METHOD PUBLIC MakeReferenceTo
VAR_INPUT
	ReferenceTarget : REFERENCE TO ETcVnThresholdType;
END_VAR
activeData REF= ReferenceTarget;
SetBaseDatatypeReference();
END_METHOD

PROPERTY PUBLIC Size : UDINT
GET
Size := SIZEOF(activeData);
END_GET
END_PROPERTY

METHOD TryMakeReferenceTo : BOOL
VAR_INPUT
	Target : I_Datatype;
END_VAR
VAR
	targetAsEnum : I_EnumDatatype;
	pTargetData : POINTER TO ETcVnThresholdType;
END_VAR
IF NOT Target.TryResolveAsEnumDatatype(targetAsEnum) THEN
	RETURN;
END_IF

IF targetAsEnum.Identifier <> Identifier THEN
	RETURN;
END_IF

pTargetData := Target.Address;
activeData REF= pTargetData^;
SetBaseDatatypeReference();
TryMakeReferenceTo := TRUE;
END_METHOD

PROPERTY PUBLIC Value : ETcVnThresholdType
GET
Value := activeData;
END_GET
SET
activeData := Value;
END_SET
END_PROPERTY

END_FUNCTION_BLOCK

// Datatypes/Enums/_ETcVnVectorCompareMethod
{attribute 'linkalways'} 
{attribute 'no_explicit_call' := 'This FB is a CLASS and must be accessed using methods or properties'}
{attribute 'enable_dynamic_creation'}
FUNCTION_BLOCK _ETcVnVectorCompareMethod EXTENDS EnumDatatypeBase
VAR
	localData : ETcVnVectorCompareMethod;
	activeData : REFERENCE TO ETcVnVectorCompareMethod;
	enumBaseDatatype : _DINT(localData);
END_VAR

METHOD FB_init : BOOL
VAR_INPUT
	bInitRetains : BOOL; // if TRUE, the retain variables are initialized (warm start / cold start)
	bInCopyCode : BOOL;  // if TRUE, the instance afterwards gets moved into the copy code (online change)
	InitialValue : ETcVnVectorCompareMethod;
END_VAR
localData := InitialValue;
AddBaseDatatype(enumBaseDatatype);
ClearReference();

AddLocalEnumeration('TCVN_VCM_EUCLIDEAN', ETcVnVectorCompareMethod.TCVN_VCM_EUCLIDEAN);
AddLocalEnumeration('TCVN_VCM_ELEMENTWISE', ETcVnVectorCompareMethod.TCVN_VCM_ELEMENTWISE);
END_METHOD

METHOD PRIVATE AddLocalEnumeration
VAR_INPUT
	Enumeration : T_MAXSTRING;
	Value : ETcVnVectorCompareMethod;
END_VAR
AddEnumeration(Enumeration, Value);
END_METHOD

METHOD IsEnumeratorValueEqual : BOOL
VAR_INPUT
	Enumerator : I_KeyValueForwardEnumerator;
END_VAR
VAR
	storedValue : ETcVnVectorCompareMethod;
END_VAR
IF NOT Enumerator.TryGet(storedValue) THEN
	RETURN;
END_IF

IsEnumeratorValueEqual := storedValue = activeData;
END_METHOD

METHOD PROTECTED SetBaseDatatypeReference
VAR_INPUT
END_VAR
enumBaseDatatype.MakeReferenceTo(activeData);
END_METHOD

PROPERTY PUBLIC Address : PVOID
GET
Address := ADR(activeData);
END_GET
END_PROPERTY

METHOD PUBLIC ClearReference
VAR_INPUT
END_VAR
activeData REF= localData;
SetBaseDatatypeReference();
END_METHOD

METHOD PUBLIC Clone : I_Datatype
VAR
    pClone : POINTER TO _ETcVnVectorCompareMethod;
END_VAR
pClone := __NEW(_ETcVnVectorCompareMethod(InitialValue := Value));
Clone := pClone^;
END_METHOD

PROPERTY PUBLIC Identifier : T_MAXSTRING
GET
Identifier := 'ETcVnVectorCompareMethod';
END_GET
END_PROPERTY

METHOD PUBLIC MakeReferenceTo
VAR_INPUT
	ReferenceTarget : REFERENCE TO ETcVnVectorCompareMethod;
END_VAR
activeData REF= ReferenceTarget;
SetBaseDatatypeReference();
END_METHOD

PROPERTY PUBLIC Size : UDINT
GET
Size := SIZEOF(activeData);
END_GET
END_PROPERTY

METHOD TryMakeReferenceTo : BOOL
VAR_INPUT
	Target : I_Datatype;
END_VAR
VAR
	targetAsEnum : I_EnumDatatype;
	pTargetData : POINTER TO ETcVnVectorCompareMethod;
END_VAR
IF NOT Target.TryResolveAsEnumDatatype(targetAsEnum) THEN
	RETURN;
END_IF

IF targetAsEnum.Identifier <> Identifier THEN
	RETURN;
END_IF

pTargetData := Target.Address;
activeData REF= pTargetData^;
SetBaseDatatypeReference();
TryMakeReferenceTo := TRUE;
END_METHOD

PROPERTY PUBLIC Value : ETcVnVectorCompareMethod
GET
Value := activeData;
END_GET
SET
activeData := Value;
END_SET
END_PROPERTY

END_FUNCTION_BLOCK

// Datatypes/Enums/_ETcVnWorldCoordinateSystem
{attribute 'linkalways'} 
{attribute 'no_explicit_call' := 'This FB is a CLASS and must be accessed using methods or properties'}
{attribute 'enable_dynamic_creation'}
FUNCTION_BLOCK _ETcVnWorldCoordinateSystem EXTENDS EnumDatatypeBase
VAR
	localData : ETcVnWorldCoordinateSystem;
	activeData : REFERENCE TO ETcVnWorldCoordinateSystem;
	enumBaseDatatype : _DINT(localData);
END_VAR

METHOD FB_init : BOOL
VAR_INPUT
	bInitRetains : BOOL; // if TRUE, the retain variables are initialized (warm start / cold start)
	bInCopyCode : BOOL;  // if TRUE, the instance afterwards gets moved into the copy code (online change)
	InitialValue : ETcVnWorldCoordinateSystem;
END_VAR
localData := InitialValue;
AddBaseDatatype(enumBaseDatatype);
ClearReference();

AddLocalEnumeration('TCVN_WCS_X_RIGHT_Y_DOWN' , ETcVnWorldCoordinateSystem.TCVN_WCS_X_RIGHT_Y_DOWN);
AddLocalEnumeration('TCVN_WCS_X_DOWN_Y_RIGHT', ETcVnWorldCoordinateSystem.TCVN_WCS_X_DOWN_Y_RIGHT);
AddLocalEnumeration('TCVN_WCS_X_LEFT_Y_DOWN', ETcVnWorldCoordinateSystem.TCVN_WCS_X_LEFT_Y_DOWN);
AddLocalEnumeration('TCVN_WCS_X_UP_Y_RIGHT', ETcVnWorldCoordinateSystem.TCVN_WCS_X_UP_Y_RIGHT);
AddLocalEnumeration('TCVN_WCS_X_RIGHT_Y_UP', ETcVnWorldCoordinateSystem.TCVN_WCS_X_RIGHT_Y_UP);
AddLocalEnumeration('TCVN_WCS_X_DOWN_Y_LEFT', ETcVnWorldCoordinateSystem.TCVN_WCS_X_DOWN_Y_LEFT);
AddLocalEnumeration('TCVN_WCS_X_LEFT_Y_UP', ETcVnWorldCoordinateSystem.TCVN_WCS_X_LEFT_Y_UP);
AddLocalEnumeration('TCVN_WCS_X_UP_Y_LEFT', ETcVnWorldCoordinateSystem.TCVN_WCS_X_UP_Y_LEFT);
END_METHOD

METHOD PRIVATE AddLocalEnumeration
VAR_INPUT
	Enumeration : T_MAXSTRING;
	Value : ETcVnWorldCoordinateSystem;
END_VAR
AddEnumeration(Enumeration, Value);
END_METHOD

METHOD IsEnumeratorValueEqual : BOOL
VAR_INPUT
	Enumerator : I_KeyValueForwardEnumerator;
END_VAR
VAR
	storedValue : ETcVnWorldCoordinateSystem;
END_VAR
IF NOT Enumerator.TryGet(storedValue) THEN
	RETURN;
END_IF

IsEnumeratorValueEqual := storedValue = activeData;
END_METHOD

METHOD PROTECTED SetBaseDatatypeReference
VAR_INPUT
END_VAR
enumBaseDatatype.MakeReferenceTo(activeData);
END_METHOD

PROPERTY PUBLIC Address : PVOID
GET
Address := ADR(activeData);
END_GET
END_PROPERTY

METHOD PUBLIC ClearReference
VAR_INPUT
END_VAR
activeData REF= localData;
SetBaseDatatypeReference();
END_METHOD

METHOD PUBLIC Clone : I_Datatype
VAR
    pClone : POINTER TO _ETcVnWorldCoordinateSystem;
END_VAR
pClone := __NEW(_ETcVnWorldCoordinateSystem(InitialValue := Value));
Clone := pClone^;
END_METHOD

PROPERTY PUBLIC Identifier : T_MAXSTRING
GET
Identifier := 'ETcVnWorldCoordinateSystem';
END_GET
END_PROPERTY

METHOD PUBLIC MakeReferenceTo
VAR_INPUT
	ReferenceTarget : REFERENCE TO ETcVnWorldCoordinateSystem;
END_VAR
activeData REF= ReferenceTarget;
SetBaseDatatypeReference();
END_METHOD

PROPERTY PUBLIC Size : UDINT
GET
Size := SIZEOF(activeData);
END_GET
END_PROPERTY

METHOD TryMakeReferenceTo : BOOL
VAR_INPUT
	Target : I_Datatype;
END_VAR
VAR
	targetAsEnum : I_EnumDatatype;
	pTargetData : POINTER TO ETcVnWorldCoordinateSystem;
END_VAR
IF NOT Target.TryResolveAsEnumDatatype(targetAsEnum) THEN
	RETURN;
END_IF

IF targetAsEnum.Identifier <> Identifier THEN
	RETURN;
END_IF

pTargetData := Target.Address;
activeData REF= pTargetData^;
SetBaseDatatypeReference();
TryMakeReferenceTo := TRUE;
END_METHOD

PROPERTY PUBLIC Value : ETcVnWorldCoordinateSystem
GET
Value := activeData;
END_GET
SET
activeData := Value;
END_SET
END_PROPERTY

END_FUNCTION_BLOCK

// Datatypes/Enums/_ETcWatchdogAccumulationType
{attribute 'linkalways'} 
{attribute 'no_explicit_call' := 'This FB is a CLASS and must be accessed using methods or properties'}
{attribute 'enable_dynamic_creation'}
FUNCTION_BLOCK _ETcWatchdogAccumulationType EXTENDS EnumDatatypeBase
VAR
	localData : ETcWatchdogAccumulationType;
	activeData : REFERENCE TO ETcWatchdogAccumulationType;
	enumBaseDatatype : _UINT(localData);
END_VAR

METHOD FB_init : BOOL
VAR_INPUT
	bInitRetains : BOOL; // if TRUE, the retain variables are initialized (warm start / cold start)
	bInCopyCode : BOOL;  // if TRUE, the instance afterwards gets moved into the copy code (online change)
	InitialValue : ETcWatchdogAccumulationType;
END_VAR
localData := InitialValue;
AddBaseDatatype(enumBaseDatatype);
ClearReference();

AddLocalEnumeration('WD_ACC_TYPE_MEAN', ETcWatchdogAccumulationType.WD_ACC_TYPE_MEAN);
AddLocalEnumeration('WD_ACC_TYPE_PRODUCT', ETcWatchdogAccumulationType.WD_ACC_TYPE_PRODUCT);
END_METHOD

METHOD PRIVATE AddLocalEnumeration
VAR_INPUT
	Enumeration : T_MAXSTRING;
	Value : ETcWatchdogAccumulationType;
END_VAR
AddEnumeration(Enumeration, Value);
END_METHOD

METHOD IsEnumeratorValueEqual : BOOL
VAR_INPUT
	Enumerator : I_KeyValueForwardEnumerator;
END_VAR
VAR
	storedValue : ETcWatchdogAccumulationType;
END_VAR
IF NOT Enumerator.TryGet(storedValue) THEN
	RETURN;
END_IF

IsEnumeratorValueEqual := storedValue = activeData;
END_METHOD

METHOD PROTECTED SetBaseDatatypeReference
VAR_INPUT
END_VAR
enumBaseDatatype.MakeReferenceTo(activeData);
END_METHOD

PROPERTY PUBLIC Address : PVOID
GET
Address := ADR(activeData);
END_GET
END_PROPERTY

METHOD PUBLIC ClearReference
VAR_INPUT
END_VAR
activeData REF= localData;
SetBaseDatatypeReference();
END_METHOD

METHOD PUBLIC Clone : I_Datatype
VAR
    pClone : POINTER TO _ETcWatchdogAccumulationType;
END_VAR
pClone := __NEW(_ETcWatchdogAccumulationType(InitialValue := Value));
Clone := pClone^;
END_METHOD

PROPERTY PUBLIC Identifier : T_MAXSTRING
GET
Identifier := 'ETcWatchdogAccumulationType';
END_GET
END_PROPERTY

METHOD PUBLIC MakeReferenceTo
VAR_INPUT
	ReferenceTarget : REFERENCE TO ETcWatchdogAccumulationType;
END_VAR
activeData REF= ReferenceTarget;
SetBaseDatatypeReference();
END_METHOD

PROPERTY PUBLIC Size : UDINT
GET
Size := SIZEOF(activeData);
END_GET
END_PROPERTY

METHOD TryMakeReferenceTo : BOOL
VAR_INPUT
	Target : I_Datatype;
END_VAR
VAR
	targetAsEnum : I_EnumDatatype;
	pTargetData : POINTER TO ETcWatchdogAccumulationType;
END_VAR
IF NOT Target.TryResolveAsEnumDatatype(targetAsEnum) THEN
	RETURN;
END_IF

IF targetAsEnum.Identifier <> Identifier THEN
	RETURN;
END_IF

pTargetData := Target.Address;
activeData REF= pTargetData^;
SetBaseDatatypeReference();
TryMakeReferenceTo := TRUE;
END_METHOD

PROPERTY PUBLIC Value : ETcWatchdogAccumulationType
GET
Value := activeData;
END_GET
SET
activeData := Value;
END_SET
END_PROPERTY

END_FUNCTION_BLOCK

// Datatypes/Enums/_GEV_CAMERA_STATE
{attribute 'linkalways'} 
{attribute 'no_explicit_call' := 'This FB is a CLASS and must be accessed using methods or properties'}
{attribute 'enable_dynamic_creation'}
FUNCTION_BLOCK _GEV_CAMERA_STATE EXTENDS EnumDatatypeBase
VAR
	localData : GEV_CAMERA_STATE;
	activeData : REFERENCE TO GEV_CAMERA_STATE;
	enumBaseDatatype : _BYTE(localData);
END_VAR

METHOD FB_init : BOOL
VAR_INPUT
	bInitRetains : BOOL; // if TRUE, the retain variables are initialized (warm start / cold start)
	bInCopyCode : BOOL;  // if TRUE, the instance afterwards gets moved into the copy code (online change)
	InitialValue : GEV_CAMERA_STATE;
END_VAR
localData := InitialValue;
AddBaseDatatype(enumBaseDatatype);
ClearReference();

AddLocalEnumeration('GEV_CAMERA_IDLE', GEV_CAMERA_STATE.GEV_CAMERA_IDLE);
AddLocalEnumeration('GEV_CONTROL_CHANNEL_OPEN_MASK', GEV_CAMERA_STATE.GEV_CONTROL_CHANNEL_OPEN_MASK);
AddLocalEnumeration('GEV_STREAM_CHANNELS_OPEN_MASK', GEV_CAMERA_STATE.GEV_STREAM_CHANNELS_OPEN_MASK);
AddLocalEnumeration('GEV_CONTROL_CHANNEL_OPEN', GEV_CAMERA_STATE.GEV_CONTROL_CHANNEL_OPEN);
AddLocalEnumeration('GEV_STREAM_CHANNELS_OPEN', GEV_CAMERA_STATE.GEV_STREAM_CHANNELS_OPEN);
END_METHOD

METHOD PRIVATE AddLocalEnumeration
VAR_INPUT
	Enumeration : T_MAXSTRING;
	Value : GEV_CAMERA_STATE;
END_VAR
AddEnumeration(Enumeration, Value);
END_METHOD

METHOD IsEnumeratorValueEqual : BOOL
VAR_INPUT
	Enumerator : I_KeyValueForwardEnumerator;
END_VAR
VAR
	storedValue : GEV_CAMERA_STATE;
END_VAR
IF NOT Enumerator.TryGet(storedValue) THEN
	RETURN;
END_IF

IsEnumeratorValueEqual := storedValue = activeData;
END_METHOD

METHOD PROTECTED SetBaseDatatypeReference
VAR_INPUT
END_VAR
enumBaseDatatype.MakeReferenceTo(activeData);
END_METHOD

PROPERTY PUBLIC Address : PVOID
GET
Address := ADR(activeData);
END_GET
END_PROPERTY

METHOD PUBLIC ClearReference
VAR_INPUT
END_VAR
activeData REF= localData;
SetBaseDatatypeReference();
END_METHOD

METHOD PUBLIC Clone : I_Datatype
VAR
    pClone : POINTER TO _GEV_CAMERA_STATE;
END_VAR
pClone := __NEW(_GEV_CAMERA_STATE(InitialValue := Value));
Clone := pClone^;
END_METHOD

PROPERTY PUBLIC Identifier : T_MAXSTRING
GET
Identifier := 'GEV_CAMERA_STATE';
END_GET
END_PROPERTY

METHOD PUBLIC MakeReferenceTo
VAR_INPUT
	ReferenceTarget : REFERENCE TO GEV_CAMERA_STATE;
END_VAR
activeData REF= ReferenceTarget;
SetBaseDatatypeReference();
END_METHOD

PROPERTY PUBLIC Size : UDINT
GET
Size := SIZEOF(activeData);
END_GET
END_PROPERTY

METHOD TryMakeReferenceTo : BOOL
VAR_INPUT
	Target : I_Datatype;
END_VAR
VAR
	targetAsEnum : I_EnumDatatype;
	pTargetData : POINTER TO GEV_CAMERA_STATE;
END_VAR
IF NOT Target.TryResolveAsEnumDatatype(targetAsEnum) THEN
	RETURN;
END_IF

IF targetAsEnum.Identifier <> Identifier THEN
	RETURN;
END_IF

pTargetData := Target.Address;
activeData REF= pTargetData^;
SetBaseDatatypeReference();
TryMakeReferenceTo := TRUE;
END_METHOD

PROPERTY PUBLIC Value : GEV_CAMERA_STATE
GET
Value := activeData;
END_GET
SET
activeData := Value;
END_SET
END_PROPERTY

END_FUNCTION_BLOCK

// Datatypes/Interface/_ITcVnImage
{attribute 'linkalways'} 
{attribute 'no_explicit_call' := 'This FB is a CLASS and must be accessed using methods or properties'}
{attribute 'enable_dynamic_creation'}
FUNCTION_BLOCK _ITcVnImage EXTENDS InterfaceDatatypeBase
VAR
	localData : ITcVnImage;
	activeData : REFERENCE TO ITcVnImage REF= localData;
END_VAR

METHOD PRIVATE TryGetElementTypeFromInfo : BOOL;
VAR_INPUT
	ImageInfo : TcVnImageInfo;
	Destination : REFERENCE TO ETcVnElementType;
END_VAR
CASE ImageInfo.stPixelFormat.nElementSize OF
	
	8 : // 8bit
	
		IF ImageInfo.stPixelFormat.bSigned THEN
			Destination := ETcVnElementType.TCVN_ET_SINT;
		ELSE	
			Destination := ETcVnElementType.TCVN_ET_USINT;
		END_IF
		TryGetElementTypeFromInfo := TRUE;
	
	16 : // 16bit
	
		IF ImageInfo.stPixelFormat.bSigned THEN
			Destination := ETcVnElementType.TCVN_ET_INT;
		ELSE	
			Destination := ETcVnElementType.TCVN_ET_UINT;
		END_IF
		TryGetElementTypeFromInfo := TRUE;
	
	32 : // 32bit
	
		IF ImageInfo.stPixelFormat.bSigned AND NOT ImageInfo.stPixelFormat.bFloat THEN
			Destination := ETcVnElementType.TCVN_ET_DINT;
			TryGetElementTypeFromInfo := TRUE;
		END_IF
		
		IF ImageInfo.stPixelFormat.bFloat THEN
			Destination := ETcVnElementType.TCVN_ET_REAL;
			TryGetElementTypeFromInfo := TRUE;
		END_IF
		
	64 : // 64bit
	
		IF ImageInfo.stPixelFormat.bFloat THEN
			Destination := ETcVnElementType.TCVN_ET_LREAL;
			TryGetElementTypeFromInfo := TRUE;
		END_IF
		
ELSE
	
	RETURN;

END_CASE
END_METHOD

PROPERTY PUBLIC Address : PVOID
GET
Address := ADR(activeData);
END_GET
END_PROPERTY

METHOD PUBLIC ClearReference
VAR_INPUT
END_VAR
activeData REF= localData;
END_METHOD

METHOD PUBLIC Clone : I_Datatype
VAR
    pClone : POINTER TO _ITcVnImage;
END_VAR
pClone := __NEW(_ITcVnImage);
Clone := pClone^;
END_METHOD

PROPERTY PUBLIC Identifier : T_MAXSTRING
GET
Identifier := 'ITcVnImage';
END_GET
END_PROPERTY

METHOD PUBLIC MakeReferenceTo
VAR_INPUT
	ReferenceTarget : REFERENCE TO ITcVnImage;
END_VAR
activeData REF= ReferenceTarget;
END_METHOD

METHOD PUBLIC SerializeWith
VAR_INPUT
	Serializer : I_Serializer;
END_VAR
VAR
	result: HRESULT;
	exportImageSize: ULINT;
	buffer : POINTER TO BYTE;
	imageInfo : _TcVnImageInfo;
END_VAR
IF NOT (activeData <> 0) THEN
	// no image available, so drop out.. need to add serialization?
	Serializer.AddNull();
	RETURN;
END_IF

result := F_VN_ExportImageSize(ipImage:=activeData, nBufferSize:=exportImageSize, hrPrev:=result);

IF FAILED(result) THEN
	// export to bmp size failed, so drop out.. need to add serialization?
	Serializer.AddNull();
	RETURN;
END_IF

IF exportImageSize > DatatypeLimits.UDINT_MAX_VALUE THEN
	// export is too big for __NEW, so drop out..
	Serializer.AddNull();
	RETURN;
END_IF

IF exportImageSize <= 0 THEN
	// export is zero size, so drop out.. 
	Serializer.AddNull();
	RETURN;
END_IF
	
buffer := __NEW(BYTE,ULINT_TO_UDINT(exportImageSize));
result := F_VN_ExportImage(ipImage:=activeData, pBuffer:=buffer, nBufferSize:=exportImageSize, hrPrev:=result);

IF FAILED(result) THEN
	// export to bmp failed, so drop out.. 
	Serializer.AddNull();
	__DELETE(buffer);
	RETURN;
END_IF

activeData.GetImageInfo(imageInfo.value);

Serializer.StartObject();
Serializer.AddKeyObject('imageInfo',imageInfo);
Serializer.AddKey('imageData');
Serializer.AddBase64(buffer,ULINT_TO_DINT(exportImageSize));
Serializer.EndObject();

__DELETE(buffer);
END_METHOD

PROPERTY PUBLIC Size : UDINT
GET
Size := SIZEOF(activeData);
END_GET
END_PROPERTY

METHOD TryDeserializeFrom : BOOL
VAR_INPUT
	Deserializer : I_Deserializer;
	Feedback : I_DeserializerFeedback;
END_VAR
VAR
	imageInfo : _TcVnImageInfo;
	imageSizeInBytes : UDINT;
	buffer : POINTER TO BYTE;
	hr : HRESULT;
	elementType : ETcVnElementType;
END_VAR
IF NOT Deserializer.TryDeserializeKeyToObject('imageInfo', imageInfo, Feedback) THEN
	RETURN;
END_IF

imageSizeInBytes := ULINT_TO_UDINT(imageInfo.nImageSize.Value);

IF imageSizeInBytes = 0 THEN
	TryDeserializeFrom := TRUE;
	RETURN;
END_IF

buffer := __NEW(BYTE, imageSizeInBytes);

IF NOT Deserializer.TryGetKeyBase64('imageData', buffer, imageSizeInBytes, Feedback) THEN
	__DELETE(buffer);
	RETURN;
END_IF

TryGetElementTypeFromInfo(imageInfo.Value, elementType);

hr := F_VN_CreateImageFromArray(
	pData := buffer,
	ipImage := activeData,
	nWidth := imageInfo.nWidth.Value,
	nHeight :=  imageInfo.nHeight.Value,
	ePixelType := elementType,
	nChannelNum := imageInfo.stPixelFormat.nChannels.Value, 
	hrPrev := hr);

__DELETE(buffer);

TryDeserializeFrom := TRUE;
END_METHOD

METHOD TryMakeReferenceTo : BOOL
VAR_INPUT
	Target : I_Datatype;
END_VAR
VAR
	targetAsInterface : I_InterfaceDatatype;
	pTargetData : POINTER TO ITcVnImage;
END_VAR
IF NOT Target.TryResolveAsInterfaceDatatype(targetAsInterface) THEN
	RETURN;
END_IF

IF targetAsInterface.Identifier <> Identifier THEN
	RETURN;
END_IF

pTargetData := Target.Address;
activeData REF= pTargetData^;
TryMakeReferenceTo := TRUE;
END_METHOD

PROPERTY PUBLIC Value : REFERENCE TO ITcVnImage
GET
Value REF= activeData;
END_GET
END_PROPERTY

END_FUNCTION_BLOCK

// Datatypes/Structs/_TcVnImageInfo
{attribute 'linkalways'} 
{attribute 'no_explicit_call' := 'This FB is a CLASS and must be accessed using methods or properties'}
{attribute 'enable_dynamic_creation'}
FUNCTION_BLOCK _TcVnImageInfo EXTENDS StructuredDatatypeBase
VAR
	localData : TcVnImageInfo;
	activeData : REFERENCE TO TcVnImageInfo REF= localData;
	_nImageSize : _ULINT(localData.nImageSize);
	_nWidth : _UDINT(localData.nWidth);
	_nHeight : _UDINT(localData.nHeight);
	_nXPadding : _UINT(localData.nXPadding);
	_nYPadding : _UINT(localData.nYPadding);
	_stPixelFormat : _TcVnPixelFormat();
END_VAR

METHOD FB_init : BOOL
VAR_INPUT
	bInitRetains : BOOL; // if TRUE, the retain variables are initialized (warm start / cold start)
	bInCopyCode : BOOL;  // if TRUE, the instance afterwards gets moved into the copy code (online change)
END_VAR
SetMemberReference();
AddMember('nImageSize',_nImageSize);
AddMember('nWidth',_nWidth);
AddMember('nHeight',_nHeight);
AddMember('nXPadding',_nXPadding);
AddMember('nYPadding',_nYPadding);
AddMember('stPixelFormat',_stPixelFormat);
END_METHOD

METHOD PROTECTED SetMemberReference
VAR_INPUT
END_VAR
_nImageSize.MakeReferenceTo(activeData.nImageSize);
_nWidth.MakeReferenceTo(activeData.nWidth);
_nHeight.MakeReferenceTo(activeData.nHeight);
_nXPadding.MakeReferenceTo(activeData.nXPadding);
_nYPadding.MakeReferenceTo(activeData.nYPadding);
_stPixelFormat.MakeReferenceTo(activeData.stPixelFormat);
END_METHOD

PROPERTY PUBLIC Address : PVOID
GET
Address := ADR(activeData);
END_GET
END_PROPERTY

METHOD PUBLIC ClearReference
VAR_INPUT
END_VAR
activeData REF= localData;
SetMemberReference();
END_METHOD

METHOD PUBLIC Clone : I_Datatype
VAR
    pClone : POINTER TO _TcVnImageInfo;
END_VAR
pClone := __NEW(_TcVnImageInfo());
pClone^.Value := Value;
Clone := pClone^;
END_METHOD

PROPERTY PUBLIC Identifier : T_MAXSTRING
GET
Identifier := 'TcVnImageInfo';
END_GET
END_PROPERTY

METHOD PUBLIC MakeReferenceTo
VAR_INPUT
	ReferenceTarget : REFERENCE TO TcVnImageInfo;
END_VAR
activeData REF= ReferenceTarget;
SetMemberReference();
END_METHOD

PROPERTY PUBLIC nHeight : Reference to _UDINT
GET
nHeight REF= _nHeight;
END_GET
END_PROPERTY

PROPERTY PUBLIC nImageSize : Reference to _ULINT
GET
nImageSize REF= _nImageSize;
END_GET
END_PROPERTY

PROPERTY PUBLIC nWidth : Reference to _UDINT
GET
nWidth REF= _nWidth;
END_GET
END_PROPERTY

PROPERTY PUBLIC nXPadding : Reference to _UINT
GET
nXPadding REF= _nXPadding;
END_GET
END_PROPERTY

PROPERTY PUBLIC nYPadding : Reference to _UINT
GET
nYPadding REF= _nYPadding;
END_GET
END_PROPERTY

PROPERTY PUBLIC Size : UDINT
GET
Size := SIZEOF(activeData);
END_GET
END_PROPERTY

PROPERTY PUBLIC stPixelFormat : Reference to _TcVnPixelFormat
GET
stPixelFormat REF= _stPixelFormat;
END_GET
END_PROPERTY

METHOD TryMakeReferenceTo : BOOL
VAR_INPUT
	Target : I_Datatype;
END_VAR
VAR
	targetAsStruct : I_StructuredDatatype;
	pTargetData : POINTER TO TcVnImageInfo;
END_VAR
IF NOT Target.TryResolveAsStructuredDatatype(targetAsStruct) THEN
	RETURN;
END_IF

IF NOT (targetAsStruct.Identifier = Identifier) THEN
	RETURN;
END_IF

pTargetData := Target.Address;
activeData REF= pTargetData^;
SetMemberReference();
TryMakeReferenceTo := TRUE;
END_METHOD

PROPERTY PUBLIC Value : reference to TcVnImageInfo
GET
Value ref= activeData;
END_GET
END_PROPERTY

END_FUNCTION_BLOCK

// Datatypes/Structs/_TcVnPixelFormat
{attribute 'linkalways'} 
{attribute 'no_explicit_call' := 'This FB is a CLASS and must be accessed using methods or properties'}
{attribute 'enable_dynamic_creation'}
FUNCTION_BLOCK _TcVnPixelFormat EXTENDS StructuredDatatypeBase
VAR
	localData : TcVnPixelFormat;
	activeData : REFERENCE TO TcVnPixelFormat REF= localData;

	_bSupported : _BIT();
	_bSigned : _BIT();
	_bPlanar : _BIT();
	_bFloat : _BIT();
	_nChannels : _BYTE(localData.nChannels);
	_ePixelEncoding : _ETcVnPixelEncoding(localData.ePixelEncoding);
	_ePixelPackMode : _ETcVnPixelPackMode(localData.ePixelPackMode);
	_nElementSize : _UINT(localData.nElementSize);
	_nTotalSize : _UINT(localData.nTotalSize);
END_VAR

METHOD FB_init : BOOL
VAR_INPUT
	bInitRetains : BOOL; // if TRUE, the retain variables are initialized (warm start / cold start)
	bInCopyCode : BOOL;  // if TRUE, the instance afterwards gets moved into the copy code (online change)
END_VAR
SetMemberReference();
AddMember('bSupported',_bSupported);
AddMember('bSigned',_bSigned);
AddMember('bPlanar',_bPlanar);
AddMember('bFloat',_bFloat);
AddMember('nChannels',_nChannels);
AddMember('ePixelEncoding',_ePixelEncoding);
AddMember('ePixelPackMode',_ePixelPackMode);
AddMember('nElementSize',_nElementSize);
AddMember('nTotalSize',_nTotalSize);
END_METHOD

METHOD PROTECTED SetMemberReference
VAR_STAT
	// this variable is used for BITADR as this function failes if used on a local variable.
	structure : TcVnPixelFormat;
END_VAR
_bSupported.MakeReferenceTo(THIS^, GetByteOffset(localData, localData.bSupported), BITADR(structure.bSupported));
_bSigned.MakeReferenceTo(THIS^, GetByteOffset(localData, localData.bSigned), BITADR(structure.bSigned));
_bPlanar.MakeReferenceTo(THIS^, GetByteOffset(localData, localData.bPlanar), BITADR(structure.bPlanar));
_bFloat.MakeReferenceTo(THIS^, GetByteOffset(localData, localData.bFloat), BITADR(structure.bFloat));
_nChannels.MakeReferenceTo(activeData.nChannels);
_ePixelEncoding.MakeReferenceTo(activeData.ePixelEncoding);
_ePixelPackMode.MakeReferenceTo(activeData.ePixelPackMode);
_nElementSize.MakeReferenceTo(activeData.nElementSize);
_nTotalSize.MakeReferenceTo(activeData.nTotalSize);
END_METHOD

PROPERTY PUBLIC Address : PVOID
GET
Address := ADR(activeData);
END_GET
END_PROPERTY

PROPERTY PUBLIC bFloat : Reference to _BIT
GET
bFloat REF= _bFloat;
END_GET
END_PROPERTY

PROPERTY PUBLIC bPlanar : Reference to _BIT
GET
bPlanar REF= _bPlanar;
END_GET
END_PROPERTY

PROPERTY PUBLIC bSigned : Reference to _BIT
GET
bSigned REF= _bSigned;
END_GET
END_PROPERTY

PROPERTY PUBLIC bSupported : Reference to _BIT
GET
bSupported REF= _bSupported;
END_GET
END_PROPERTY

METHOD PUBLIC ClearReference
VAR_INPUT
END_VAR
activeData REF= localData;
SetMemberReference();
END_METHOD

METHOD PUBLIC Clone : I_Datatype
VAR
    pClone : POINTER TO _TcVnPixelFormat;
END_VAR
pClone := __NEW(_TcVnPixelFormat());
pClone^.Value := Value;
Clone := pClone^;
END_METHOD

PROPERTY PUBLIC ePixelEncoding : Reference to _ETcVnPixelEncoding
GET
ePixelEncoding REF= _ePixelEncoding;
END_GET
END_PROPERTY

PROPERTY PUBLIC ePixelPackMode : Reference to _ETcVnPixelPackMode
GET
ePixelPackMode REF= _ePixelPackMode;
END_GET
END_PROPERTY

PROPERTY PUBLIC Identifier : T_MAXSTRING
GET
Identifier := 'TcVnPixelFormat';
END_GET
END_PROPERTY

METHOD PUBLIC MakeReferenceTo
VAR_INPUT
	ReferenceTarget : REFERENCE TO TcVnPixelFormat;
END_VAR
activeData REF= ReferenceTarget;
SetMemberReference();
END_METHOD

PROPERTY PUBLIC nChannels : Reference to _BYTE
GET
nChannels REF= _nChannels;
END_GET
END_PROPERTY

PROPERTY PUBLIC nElementSize : Reference to _UINT
GET
nElementSize REF= _nElementSize;
END_GET
END_PROPERTY

PROPERTY PUBLIC nTotalSize : Reference to _UINT
GET
nTotalSize REF= _nTotalSize;
END_GET
END_PROPERTY

PROPERTY PUBLIC Size : UDINT
GET
Size := SIZEOF(activeData);
END_GET
END_PROPERTY

METHOD TryMakeReferenceTo : BOOL
VAR_INPUT
	Target : I_Datatype;
END_VAR
VAR
	targetAsStruct : I_StructuredDatatype;
	pTargetData : POINTER TO TcVnPixelFormat;
END_VAR
IF NOT Target.TryResolveAsStructuredDatatype(targetAsStruct) THEN
	RETURN;
END_IF

IF NOT (targetAsStruct.Identifier = Identifier) THEN
	RETURN;
END_IF

pTargetData := Target.Address;
activeData REF= pTargetData^;
SetMemberReference();
TryMakeReferenceTo := TRUE;
END_METHOD

PROPERTY PUBLIC Value : reference to TcVnPixelFormat
GET
Value REF= activeData;
END_GET
END_PROPERTY

END_FUNCTION_BLOCK

// Datatypes/VisionDatatypePack
{attribute 'linkalways'} 
{attribute 'no_explicit_call' := 'This FB is a CLASS and must be accessed using methods or properties'}
{attribute 'enable_dynamic_creation'}
FUNCTION_BLOCK VisionDatatypePack IMPLEMENTS I_DatatypePack
VAR
	// alias
	
	// enums
	_eTcVn2dCodeSearchStrategy : _ETcVn2dCodeSearchStrategy(ETcVn2dCodeSearchStrategy.TCVN_CSS_DEFAULT);
	
	// structures
	_tcVnImageInfo : _TcVnImageInfo;
	_tcVnPixelFormat : _TcVnPixelFormat;
	
	// interface
	_iTcVnImage : _ITcVnImage;
	
END_VAR

METHOD RegisterWithDatatypes
VAR_INPUT
	Datatypes : I_Datatypes;
END_VAR
// enums
Datatypes.RegisterDatatype(_eTcVn2dCodeSearchStrategy);

// structures
Datatypes.RegisterDatatype(_tcVnImageInfo);
Datatypes.RegisterDatatype(_tcVnPixelFormat);

// interfaces
Datatypes.RegisterDatatype(_iTcVnImage);
END_METHOD

END_FUNCTION_BLOCK

// Nodes/VisionNodePack
{attribute 'linkalways'} 
{attribute 'no_explicit_call' := 'This FB is a CLASS and must be accessed using methods or properties'}
{attribute 'enable_dynamic_creation'}
FUNCTION_BLOCK VisionNodePack IMPLEMENTS I_NodePack
VAR
	//node : Node;
END_VAR

METHOD PUBLIC RegisterWithNodeFactory
VAR_INPUT
	NodeFactory : I_NodeFactory;
END_VAR
//NodeFactory.AddNodeAsPrototype('Vision/Node',Node);
END_METHOD

END_FUNCTION_BLOCK

// VisionPack
{attribute 'linkalways'} 
{attribute 'no_explicit_call' := 'This FB is a CLASS and must be accessed using methods or properties'}
{attribute 'enable_dynamic_creation'}
FUNCTION_BLOCK VisionPack IMPLEMENTS I_GraphPack
VAR
	visionDatatypePack : VisionDatatypePack;
	visionNodePack : VisionNodePack;
END_VAR

METHOD RegisterWithDatatypes
VAR_INPUT
	Datatypes : I_Datatypes;
END_VAR
visionDatatypePack.RegisterWithDatatypes(Datatypes);
END_METHOD

METHOD PUBLIC RegisterWithNodeFactory
VAR_INPUT
	NodeFactory : I_NodeFactory;
END_VAR
visionNodePack.RegisterWithNodeFactory(NodeFactory);
END_METHOD

END_FUNCTION_BLOCK
